(* CODESYS project METS_Software_Library.library
   Company: Marden Edwards LTD
   DefaultNamespace: LibB
   LanguageModelAttribute: qualified-access-only
   Title: METS_Software_Library
   Placeholder: LibA
   Version: 0.0.1

Project tree, tasks and I/O mapping:
  libraries: Tc2_Standard, * (Beckhoff Automation GmbH); Tc2_System, * (Beckhoff Automation GmbH); Tc2_Utilities, * (Beckhoff Automation GmbH)
  Maths/
    function F_Add [ST]
  Strings/
    Alias/
      data type T_Char
      data type T_LONGString
    Concat/
      function F_STRING_Concat3 [ST]
      function F_STRING_Concat4 [ST]
      function F_STRING_Concat5 [ST]
      function F_STRING_Concat6 [ST]
      function F_STRING_Concat7 [ST]
      function F_STRING_Concat8 [ST]
      function F_STRING_Concat9 [ST]
      function F_STRING_LongCONCAT [ST]
    Enumerations/
      data type E_STRING_ValidationCode
    Extract/
      function block FB_STRING_Extract [ST]
      function block FB_STRING_Extract_V2 [ST]
      function block FB_STRING_ExtractLong [ST]
    Manipulation/
      function F_STRING_AddPadding [ST]
      function F_STRING_AddPrefix [ST]
      function F_STRING_AddSuffix [ST]
      function F_STRING_CodeToHex [ST]
      function F_STRING_LongDELETE [ST]
      function F_STRING_LongFIND [ST]
      function F_STRING_LongLEFT [ST]
      function F_STRING_LongMID [ST]
      function F_STRING_LongRIGHT [ST]
      function F_STRING_ReplaceSingleChar [ST]
      function F_STRING_Wildcard [ST]
      function F_STRING_WriteEscapeCharacters [ST]
    Validation/
      function F_STRING_InvalidateASCIIChar [ST]
      function F_STRING_InvalidateNumericChar [ST]
      function F_STRING_IsNumber [ST]
      function F_STRING_Validate [ST]
      function F_STRING_ValidateCode [ST]
*)

// Strings/Alias/T_Char
TYPE T_Char : STRING(1); END_TYPE

// Strings/Alias/T_LONGString
TYPE T_LONGString : STRING(1024); END_TYPE

// Strings/Enumerations/E_STRING_ValidationCode
{attribute 'qualified_only'}
{attribute 'strict'}
{attribute 'to_string'}
TYPE E_STRING_ValidationCode :
(
	VALID := 0,
	EMPTY_STRING := 1,
	TOO_SHORT := 2,
	TOO_LONG := 3,
	INVALID := 4,
	INVALID_DECIMALPOINT := 5,
	MAXIMUM_LENGTH_EXCEEDED := 6
);
END_TYPE

// Maths/F_Add
FUNCTION F_Add : INT
VAR_INPUT
    nValue1 : INT;
    nValue2 : INT;
END_VAR

F_Add := nValue1 + nValue2;

END_FUNCTION

// Strings/Concat/F_STRING_Concat3
(* concatenate 3 strings *)
FUNCTION F_STRING_Concat3 : T_MaxString
VAR_INPUT
	sString1			: T_MaxString;		(* first string *)
	sString2			: T_MaxString;		(* second string *)
	sString3			: T_MaxString;		(* third string *)
END_VAR
VAR
END_VAR

F_STRING_Concat3 := CONCAT(sString1, sString2);
F_STRING_Concat3 := CONCAT(F_STRING_Concat3, sString3);

END_FUNCTION

// Strings/Concat/F_STRING_Concat4
(* concatenate 4 strings *)
FUNCTION F_STRING_Concat4 : T_MaxString
VAR_INPUT
	sString1			: T_MaxString;		(* first string *)
	sString2			: T_MaxString;		(* second string *)
	sString3			: T_MaxString;		(* third string *)
	sString4			: T_MaxString;		(* fourth string *)
END_VAR
VAR
END_VAR

F_STRING_Concat4 := CONCAT(sString1, sString2);
F_STRING_Concat4 := CONCAT(F_STRING_Concat4, sString3);
F_STRING_Concat4 := CONCAT(F_STRING_Concat4, sString4);

END_FUNCTION

// Strings/Concat/F_STRING_Concat5
(* concatenate 5 strings *)
FUNCTION F_STRING_Concat5 : T_MaxString
VAR_INPUT
	sString1			: T_MaxString;		(* first string *)
	sString2			: T_MaxString;		(* second string *)
	sString3			: T_MaxString;		(* third string *)
	sString4			: T_MaxString;		(* fourth string *)
	sString5			: T_MaxString;		(* fifth string *)
END_VAR
VAR
END_VAR

F_STRING_Concat5 := CONCAT(sString1, sString2);
F_STRING_Concat5 := CONCAT(F_STRING_Concat5, sString3);
F_STRING_Concat5 := CONCAT(F_STRING_Concat5, sString4);
F_STRING_Concat5 := CONCAT(F_STRING_Concat5, sString5);

END_FUNCTION

// Strings/Concat/F_STRING_Concat6
(* concatenate 6 strings *)
FUNCTION F_STRING_Concat6 : T_MaxString
VAR_INPUT
	sString1			: T_MaxString;		(* first string *)
	sString2			: T_MaxString;		(* second string *)
	sString3			: T_MaxString;		(* third string *)
	sString4			: T_MaxString;		(* fourth string *)
	sString5			: T_MaxString;		(* fifth string *)
	sString6			: T_MaxString;		(* sixth string *)
END_VAR
VAR
END_VAR

F_STRING_Concat6 := CONCAT(sString1, sString2);
F_STRING_Concat6 := CONCAT(F_STRING_Concat6, sString3);
F_STRING_Concat6 := CONCAT(F_STRING_Concat6, sString4);
F_STRING_Concat6 := CONCAT(F_STRING_Concat6, sString5);
F_STRING_Concat6 := CONCAT(F_STRING_Concat6, sString6);

END_FUNCTION

// Strings/Concat/F_STRING_Concat7
(* concatenate 7 strings *)
FUNCTION F_STRING_Concat7 : T_MaxString
VAR_INPUT
	sString1			: T_MaxString;		(* first string *)
	sString2			: T_MaxString;		(* second string *)
	sString3			: T_MaxString;		(* third string *)
	sString4			: T_MaxString;		(* fourth string *)
	sString5			: T_MaxString;		(* fifth string *)
	sString6			: T_MaxString;		(* sixth string *)
	sString7			: T_MaxString;		(* seventh string *)
END_VAR
VAR
END_VAR

F_STRING_Concat7 := CONCAT(sString1, sString2);
F_STRING_Concat7 := CONCAT(F_STRING_Concat7, sString3);
F_STRING_Concat7 := CONCAT(F_STRING_Concat7, sString4);
F_STRING_Concat7 := CONCAT(F_STRING_Concat7, sString5);
F_STRING_Concat7 := CONCAT(F_STRING_Concat7, sString6);
F_STRING_Concat7 := CONCAT(F_STRING_Concat7, sString7);

END_FUNCTION

// Strings/Concat/F_STRING_Concat8
(* concatenate 8 strings *)
FUNCTION F_STRING_Concat8 : T_MaxString
VAR_INPUT
	sString1			: T_MaxString;		(* first string *)
	sString2			: T_MaxString;		(* second string *)
	sString3			: T_MaxString;		(* third string *)
	sString4			: T_MaxString;		(* fourth string *)
	sString5			: T_MaxString;		(* fifth string *)
	sString6			: T_MaxString;		(* sixth string *)
	sString7			: T_MaxString;		(* seventh string *)
	sString8			: T_MaxString;		(* eigth string *)
END_VAR
VAR
END_VAR

F_STRING_Concat8 := CONCAT(sString1, sString2);
F_STRING_Concat8 := CONCAT(F_STRING_Concat8, sString3);
F_STRING_Concat8 := CONCAT(F_STRING_Concat8, sString4);
F_STRING_Concat8 := CONCAT(F_STRING_Concat8, sString5);
F_STRING_Concat8 := CONCAT(F_STRING_Concat8, sString6);
F_STRING_Concat8 := CONCAT(F_STRING_Concat8, sString7);
F_STRING_Concat8 := CONCAT(F_STRING_Concat8, sString8);

END_FUNCTION

// Strings/Concat/F_STRING_Concat9
(* concatenate 9 strings *)
FUNCTION F_STRING_Concat9 : T_MaxString
VAR_INPUT
	sString1			: T_MaxString;		(* first string *)
	sString2			: T_MaxString;		(* second string *)
	sString3			: T_MaxString;		(* third string *)
	sString4			: T_MaxString;		(* fourth string *)
	sString5			: T_MaxString;		(* fifth string *)
	sString6			: T_MaxString;		(* sixth string *)
	sString7			: T_MaxString;		(* seventh string *)
	sString8			: T_MaxString;		(* eigth string *)
	sString9			: T_MaxString;		(* ninth string *)
END_VAR
VAR
END_VAR
(*
-------------------------------------------------------------------------------------------------
Date		Version	Author	Comments
-------------------------------------------------------------------------------------------------
30/01/2015	3.00.00	PB		No change

-------------------------------------------------------------------------------------------------
05/02/2010	1.00.00	PB		Initial release

-------------------------------------------------------------------------------------------------
*)

F_STRING_Concat9 := CONCAT(sString1, sString2);
F_STRING_Concat9 := CONCAT(F_STRING_Concat9, sString3);
F_STRING_Concat9 := CONCAT(F_STRING_Concat9, sString4);
F_STRING_Concat9 := CONCAT(F_STRING_Concat9, sString5);
F_STRING_Concat9 := CONCAT(F_STRING_Concat9, sString6);
F_STRING_Concat9 := CONCAT(F_STRING_Concat9, sString7);
F_STRING_Concat9 := CONCAT(F_STRING_Concat9, sString8);
F_STRING_Concat9 := CONCAT(F_STRING_Concat9, sString9);

END_FUNCTION

// Strings/Concat/F_STRING_LongCONCAT
(* concatenate function for long strings *)
FUNCTION F_STRING_LongCONCAT : T_LongSTRING
VAR_INPUT
	sString1			: T_LongSTRING;		(* first string *)
	sString2			: T_LongSTRING;		(* second string *)
END_VAR
VAR
	_pPointer			: POINTER TO T_LongSTRING;		
	_nString1Length		: UINT;
	_nString2Length		: UINT;
END_VAR

(* length of 1st input string *)
_pPointer := ADR(sString1);
_nString1Length := TO_UINT(LEN2(_pPointer));

_pPointer := ADR(sString2);
(* max length of 2nd input string that can be handled without exceeding length of output string *)
_nString2Length := MIN(TO_UINT(LEN2(_pPointer)), SIZEOF(F_STRING_LongCONCAT) - _nString1Length - 1);

(* output string length <= 255 chars *)
IF _nString1Length + _nString2Length <= 255 THEN

	F_STRING_LongCONCAT := CONCAT(sString1, sString2);

(* output string length > 255 chars *)
ELSE

	(* string length > 0, must not call MEMMOVE with 0 bytes *)
	IF _nString1Length > 0 THEN

		(* move strString1 to output string *)
		MEMMOVE(ADR(F_STRING_LongCONCAT), ADR(sString1), _nString1Length);
		
	END_IF

	(* string length > 0, must not call MEMMOVE with 0 bytes *)
	IF _nString2Length > 0 THEN

		(* move strString2 to output string, clamp output if final length of string exceeds T_LongSTRING *)
		MEMMOVE(ADR(F_STRING_LongCONCAT) + _nString1Length, ADR(sString2), _nString2Length);
		
	END_IF

	(* reset last char to 16#00 to terminate the string with NULL *)
	MEMSET(ADR(F_STRING_LongCONCAT) + _nString1Length + _nString2Length, 16#00, 1);
	
END_IF

END_FUNCTION

// Strings/Extract/FB_STRING_Extract
(* extracts a substring defined by prefix and suffix *)
FUNCTION_BLOCK FB_STRING_Extract
VAR_INPUT
	bExtractData			: BOOL;			(* set TRUE to remove prefix and suffix from strData *)
	nExtractCharacters		: UINT;			(* if suffix is blank, number of data chars to extract *)
	sPrefix					: T_MaxString;	(* prefix string *)
	sSuffix					: T_MaxString;	(* suffix string *)
END_VAR
VAR_IN_OUT
	sString					: T_MaxString;	(* string to be searched *)
END_VAR
VAR_OUTPUT
	bStringFound			: BOOL;			(* TRUE = sub-string with matching prefix/suffix found *)
	nStartPosition			: UINT;			(* start pos of extracted string in sString *)
	sExtractedCharacters	: T_MaxString;	(* extracted data *)
END_VAR
VAR
	_nStringLength			: UINT;
	_nPrefixLength			: UINT;
	_nSuffixLength			: UINT;
	_nEndPosition			: UINT;
	_bStartPositionFound	: BOOL;
	_bEndPositionFound		: BOOL;
	_nCharacters			: UINT;
	_nMaxIndex				: UINT;
	_nIndex					: UINT;
END_VAR

(* calc string lengths *)
_nStringLength := INT_TO_UINT(LEN(sString));
_nPrefixLength := INT_TO_UINT(LEN(sPrefix));
_nSuffixLength := INT_TO_UINT(LEN(sSuffix));

(* string to be searched is not empty and prefix or suffix or no or chars to extract is defined *)
IF _nStringLength > 0 AND (_nPrefixLength > 0 OR _nSuffixLength > 0 OR nExtractCharacters > 0) THEN

	(* clear outputs *)
	bStringFound := FALSE;
	_nCharacters := 0;
	nStartPosition := 0;
	sExtractedCharacters := '';

	(* initialise char index values *)
	_bStartPositionFound := FALSE;
	_bEndPositionFound := FALSE;
	_nEndPosition := 0;

	(* max search index, based on string length - 1 due to starting at 0 and length of prefix *)
	_nMaxIndex := (_nStringLength - 1) + (_nPrefixLength - 1);

	(* for each character in the string *)
	FOR _nIndex := 0 TO _nMaxIndex DO

		(* prefix has not been found *)
		IF _bStartPositionFound = FALSE THEN

			(* no prefix defined  *)
			IF _nPrefixLength = 0 THEN

				(* start at beginning if string *)
				nStartPosition := 1;
				_bStartPositionFound := TRUE;

			(* prefix defined  *)
			ELSE

				(* compare partial string with prefix *)
				IF MEMCMP(ADR(sString) + _nIndex, ADR(sPrefix), _nPrefixLength) = 0 THEN

					(* prefix position found *)
					nStartPosition := _nIndex + 1;
					_bStartPositionFound := TRUE;

					(* skip to end of prefix to continue search *)
					_nIndex := _nIndex + _nPrefixLength - 1;
					
				END_IF
				
			END_IF

		(* suffix has not been found *)
		ELSIF _bEndPositionFound = FALSE THEN

			(* no suffix defined  *)
			IF _nSuffixLength = 0 THEN

				(* start at 1st char of string *)
				_bEndPositionFound := TRUE;

				(* calculate end position *)
				_nEndPosition := MIN((nStartPosition - 1) + nExtractCharacters + _nPrefixLength, _nStringLength);

			(* suffix defined  *)
			ELSE

				(* compare partial string with suffix *)
				IF MEMCMP(ADR(sString) + _nIndex, ADR(sSuffix), _nSuffixLength) = 0 THEN

					(* suffix position found, calculate end position *)
					_nEndPosition := _nIndex + _nSuffixLength;
					_bEndPositionFound := TRUE;

					(* no prefix defined and number of chars to extract is defined *)
					IF _nPrefixLength = 0 AND nExtractCharacters > 0 THEN

						(* re-calculate start position *)
						nStartPosition := MAX(_nEndPosition - nExtractCharacters - 1, 1);
						
					END_IF

					(* search complete, quit FOR loop *)
					EXIT;
					
				END_IF
				
			END_IF

		(* prefix and suffix found *)
		ELSE

			(* quit FOR loop *)
			EXIT;
			
		END_IF
		
	END_FOR

	(* start and end positions known *)
	IF _bStartPositionFound = TRUE AND _bEndPositionFound = TRUE THEN

		(* string has been found *)
		bStringFound := TRUE;

		(* return string without prefix and suffix *)
		IF bExtractData = TRUE THEN

			(* total chars to be moved to strData *)
			_nCharacters := (_nEndPosition - (nStartPosition - 1)) - _nPrefixLength - _nSuffixLength;

			(* 1 or more chars to be moved *)
			IF _nCharacters > 0 THEN

				(* move data to sResult *)
				MEMMOVE(ADR(sExtractedCharacters), ADR(sString) + (nStartPosition - 1) + _nPrefixLength, _nCharacters);
				
			END_IF

		(* return string with prefix and suffix *)
		ELSE

			(* total chars to be moved to strData *)
			_nCharacters := _nEndPosition - (nStartPosition - 1);

			(* 1 or more chars to be moved *)
			IF _nCharacters > 0 THEN

				(* move data to sResult *)
				MEMMOVE(ADR(sExtractedCharacters), ADR(sString) + (nStartPosition - 1), _nCharacters);
				
			END_IF
			
		END_IF

		(* terminate sResult *)
		MEMSET(ADR(sExtractedCharacters) + _nCharacters, 16#00, 1);

		(* 1 or more chars after strSuffix *)
		IF _nStringLength > (_nEndPosition - (nStartPosition - 1)) THEN

			(* shift post-suffix chars to prefix position *)
			MEMMOVE(ADR(sString) + (nStartPosition - 1), ADR(sString) + _nEndPosition, _nStringLength - (_nEndPosition - (nStartPosition - 1)));
			
		END_IF

		(* terminate strString *)
		MEMSET(ADR(sString) + _nStringLength - (_nEndPosition - (nStartPosition - 1)), 16#00, 1);
		
	END_IF

(* string to be searched is empty or prefix and suffix and both blank *)
ELSE

	(* clear outputs *)
	bStringFound := FALSE;
	_nCharacters := 0;
	sExtractedCharacters := '';
	
END_IF

END_FUNCTION_BLOCK

// Strings/Extract/FB_STRING_Extract_V2
(* extracts a substring defined by prefix and suffix *)
FUNCTION_BLOCK FB_STRING_Extract_V2
VAR_INPUT
	bIgnoreCase				: BOOL;
	sPrefix					: STRING(10);	(* prefix string *)
	sSuffix					: STRING(10);	(* suffix string *)
	nExtractCharacters		: BYTE;			(* if suffix is blank, >0 = no of chars to extract , 0 = remainder of string *)
END_VAR
VAR_IN_OUT
	sString					: T_MaxString;	(* string to be searched *)
END_VAR
VAR_OUTPUT
	bStringFound			: BOOL;			(* TRUE = sub-string with matching prefix/suffix found *)
	nCharactersFound		: UINT;			(* no of chars in sub-string *)
	sExtractedCharacters	: T_MaxString;	(* sub-string with prefix and suffix *)
END_VAR
VAR
	_nPrefixPosition		: UINT;
	_nSuffixPosition		: UINT;
	_nIndex					: UINT;
	_sStringInternal		: T_MaxString;
	_sPrefixInternal		: STRING(10);
	_sSuffixInternal		: STRING(10);
	_sCheckString			: STRING(10);
END_VAR

(* string to be searched is not empty *)
IF LEN(sString) > 0 THEN

	(* matching for Prefix and Suffix is case-sesnsitive *)
	IF bIgnoreCase = FALSE THEN

		(* internal comparators are not changed *)
		_sStringInternal := sString;
		_sPrefixInternal := sPrefix;
		_sSuffixInternal := sSuffix;

	(* ignore case when matching for Prefix and Suffix *)
	ELSE

		(* internal comparators are all converted to lower case *)
		_sStringInternal := F_ToLCase(sString);
		_sPrefixInternal := F_ToLCase(sPrefix);
		_sSuffixInternal := F_ToLCase(sSuffix);
		
	END_IF

	(* prefix is blank *)
	IF _sPrefixInternal = '' THEN

		(* start at beginning of string *)
		_nPrefixPosition := 1;

	(* prefix is not blank *)
	ELSE

		(* find 1st occurrence of prefix in strString *)
		_nPrefixPosition := FIND(_sStringInternal, _sPrefixInternal);
		
	END_IF

	(* suffix is blank *)
	IF _sSuffixInternal = '' THEN
	
		(* no of chars not specified *)
		IF nExtractCharacters = 0 THEN
	
			(* finish at end of string *)
			_nSuffixPosition := LEN(_sStringInternal);
	
		(* no of chars specified *)
		ELSE
	
			(* finish at end of string *)
			_nSuffixPosition := _nPrefixPosition + nExtractCharacters - 1;
			
		END_IF
	
	(* suffix is not blank *)
	ELSE
	
		_nSuffixPosition := 0;
	
		(* find 1st occurrence of suffix in strString AFTER position of strPrefix *)
		FOR _nIndex := _nPrefixPosition + LEN(_sPrefixInternal) TO LEN(_sStringInternal) DO
	
			(* extract string same length as suffix string *)
			_sCheckString := MID(_sStringInternal, LEN(_sSuffixInternal), _nIndex);
	
			(* extracted string = suffix string *)
			IF _sCheckString = _sSuffixInternal THEN
	
				(* position of suffix string *)
				_nSuffixPosition := _nIndex;
				EXIT;
				
			END_IF
			
		END_FOR
		
	END_IF
	
	
	(* prefix and suffix both exist *)
	IF _nPrefixPosition > 0 AND _nSuffixPosition > 0 THEN
	
		(* extract sub-string *)
		sExtractedCharacters := MID(sString, _nSuffixPosition + MAX(LEN(_sSuffixInternal), 1) - _nPrefixPosition, _nPrefixPosition);

		(* delete sub-string *)
		sString := DELETE(sString, _nSuffixPosition + MAX(LEN(_sSuffixInternal), 1) - _nPrefixPosition, _nPrefixPosition);
	
		(* update outputs *)
		bStringFound := TRUE;
		nCharactersFound := LEN(sExtractedCharacters);
	
	(* no prefix or suffix defined, cannot search for string *)
	ELSE
	
		sExtractedCharacters := '';
		bStringFound := FALSE;
		nCharactersFound := 0;
		
	END_IF

(* string to be searched is empty *)
ELSE

	(* reset outputs *)
	bStringFound := FALSE;
	nCharactersFound := 0;
	sExtractedCharacters := '';
	
END_IF

END_FUNCTION_BLOCK

// Strings/Extract/FB_STRING_ExtractLong
(* extracts a substring from a long string defined by prefix and suffix *)
FUNCTION_BLOCK FB_STRING_ExtractLong
VAR_INPUT
	bExtractData			: BOOL;			(* set TRUE to remove prefix and suffix from strData *)
	nExtractCharacters		: UINT;			(* if suffix is blank, number of data chars to extract *)
	sPrefix					: T_MaxString;	(* prefix string *)
	sSuffix					: T_MaxString;	(* suffix string *)
END_VAR
VAR_IN_OUT
	sString					: T_LongSTRING;	(* string to be searched *)
END_VAR
VAR_OUTPUT
	bStringFound			: BOOL;			(* TRUE = sub-string with matching prefix/suffix found *)
	nStartPosition			: UINT;			(* start pos of extracted string in strString *)
	sExtractedCharacters	: T_LongSTRING;	(* extracted data *)
END_VAR
VAR
	_bStartPositionFound	: BOOL;
	_bEndPositionFound		: BOOL;
	_nStringLength			: UINT;
	_nPrefixLength			: UINT;
	_nSuffixLength			: UINT;
	_nEndPosition			: UINT;
	_nCharacters			: UINT;
	_nMaxIndex				: UINT;
	_nIndex					: UINT;
END_VAR

(* calc string lengths *)
_nStringLength := UDINT_TO_UINT(LEN2(ADR(sString)));
_nPrefixLength := INT_TO_UINT(LEN(sPrefix));
_nSuffixLength := INT_TO_UINT(LEN(sSuffix));

(* string to be searched is not empty and prefix or suffix or no or chars to extract is defined *)
IF _nStringLength > 0 AND (_nPrefixLength > 0 OR _nSuffixLength > 0 OR nExtractCharacters > 0) THEN

	(* clear outputs *)
	bStringFound := FALSE;
	_nCharacters := 0;
	nStartPosition := 0;
	sExtractedCharacters := '';

	(* initialise char index values *)
	_bStartPositionFound := FALSE;
	_bEndPositionFound := FALSE;
	_nEndPosition := 0;

	(* max search index, based on string length - 1 due to starting at 0 and length of prefix *)
	_nMaxIndex := (_nStringLength - 1) + (_nPrefixLength - 1);

	(* for each character in the string *)
	FOR _nIndex := 0 TO _nMaxIndex DO

		(*IF nIndex = nMaxIndex  AND NOT bStartPosFound THEN

			strString :='1';

		(* prefix has not been found *)
		ELS*)IF _bStartPositionFound = FALSE THEN

			(* no prefix defined  *)
			IF _nPrefixLength = 0 THEN

				(* start at beginning if string *)
				nStartPosition := 1;
				_bStartPositionFound := TRUE;

			(* prefix defined  *)
			ELSE

				(* compare partial string with prefix *)
				IF MEMCMP(ADR(sString) + _nIndex, ADR(sPrefix), _nPrefixLength) = 0 THEN

					(* prefix position found *)
					nStartPosition := _nIndex + 1;
					_bStartPositionFound := TRUE;

					(* skip to end of prefix to continue search *)
					_nIndex := _nIndex + _nPrefixLength - 1;
					
				END_IF
				
			END_IF

		(* suffix has not been found *)
		ELSIF _bEndPositionFound = FALSE THEN

			(* no suffix defined  *)
			IF _nSuffixLength = 0 THEN

				(* start at 1st char of string *)
				_bEndPositionFound := TRUE;

				(* calculate end position *)
				_nEndPosition := MIN((nStartPosition - 1) + nExtractCharacters + _nPrefixLength, _nStringLength);

			(* suffix defined  *)
			ELSE

				(* compare partial string with suffix *)
				IF MEMCMP(ADR(sString) + _nIndex, ADR(sSuffix), _nSuffixLength) = 0 THEN

					(* suffix position found, calculate end position *)
					_nEndPosition := _nIndex + _nSuffixLength;
					_bEndPositionFound := TRUE;

					(* no prefix defined and number of chars to extract is defined *)
					IF _nPrefixLength = 0 AND nExtractCharacters > 0 THEN

						(* re-calculate start position *)
						nStartPosition := MAX(_nEndPosition - nExtractCharacters - 1, 1);
						
					END_IF

					(* search complete, quit FOR loop *)
					EXIT;
					
				END_IF
				
			END_IF

		(* prefix and suffix found *)
		ELSE

			(* quit FOR loop *)
			EXIT;

		END_IF
		
	END_FOR

	(* start and end positions known *)
	IF _bStartPositionFound = TRUE AND _bEndPositionFound = TRUE THEN

		(* string has been found *)
		bStringFound := TRUE;

		(* return string without prefix and suffix *)
		IF bExtractData = TRUE THEN

			(* total chars to be moved to strData *)
			_nCharacters := (_nEndPosition - (nStartPosition - 1)) - _nPrefixLength - _nSuffixLength;

			(* 1 or more chars to be moved *)
			IF _nCharacters > 0 THEN

				(* move data to strData *)
				MEMMOVE(ADR(sExtractedCharacters), ADR(sString) + (nStartPosition - 1) + _nPrefixLength, _nCharacters);
				
			END_IF

		(* return string with prefix and suffix *)
		ELSE

			(* total chars to be moved to strData *)
			_nCharacters := _nEndPosition - (nStartPosition - 1);

			(* 1 or more chars to be moved *)
			IF _nCharacters > 0 THEN

				(* move data to strData *)
				MEMMOVE(ADR(sExtractedCharacters), ADR(sString) + (nStartPosition - 1), _nCharacters);
				
			END_IF
			
		END_IF

		(* terminate strData *)
		MEMSET(ADR(sExtractedCharacters) + _nCharacters, 16#00, 1);

		(* 1 or more chars after strSuffix *)
		IF _nStringLength> (_nEndPosition - (nStartPosition - 1)) THEN

			(* shift post-suffix chars to prefix position *)
			MEMMOVE(ADR(sString) + (nStartPosition - 1), ADR(sString) + _nEndPosition, _nStringLength - (_nEndPosition - (nStartPosition - 1)));
			
		END_IF

		(* terminate strString *)
		MEMSET(ADR(sString) + _nStringLength - (_nEndPosition - (nStartPosition - 1)), 16#00, 1);
		
	END_IF

(* string to be searched is empty or prefix and suffix and both blank *)
ELSE

	(* clear outputs *)
	bStringFound := FALSE;
	_nCharacters := 0;
	sExtractedCharacters := '';
	
END_IF

END_FUNCTION_BLOCK

// Strings/Manipulation/F_STRING_AddPadding
(* Adds leading '0' to a given string returning it as a string.  Number has to be a positive integer *)
FUNCTION F_STRING_AddPadding : STRING 		(* String with leading '0' applied.  Max length 80 characters *)
VAR_INPUT
	nNumber				: UDINT;			(* Number to add leading '0' to *)
	nSize				: UINT;				(* Total size of the returning string including the original number *)
END_VAR
VAR
	_Size				: UINT;
	_sTemp				: STRING;
END_VAR

IF nSize > 80 THEN 

	_sTemp := UDINT_TO_STRING(nNumber);
	F_STRING_AddPadding := _sTemp;

ELSE

	_Size := nSize;
	_sTemp := UDINT_TO_STRING(nNumber);
	
	WHILE LEN(_sTemp) < _Size DO

		_sTemp := CONCAT('0',_sTemp);

	END_WHILE
	
	F_STRING_AddPadding := _sTemp;

END_IF

END_FUNCTION

// Strings/Manipulation/F_STRING_AddPrefix
(* add specified char(s) in front of a string to make up to specified length *)
FUNCTION F_STRING_AddPrefix : T_MaxString
VAR_INPUT
	sString				: T_MaxString;	(* initial string *)
	nTargetLength 		: UINT;			(* total string length required *)
	sCharacterToAppend	: T_Char;		(* character to be inserted at start of the string *)
END_VAR
VAR
	_nStringLength		: UINT;
	_nCharactersRequired: UINT; 
END_VAR

(* length of input string *)
_nStringLength := TO_UINT(LEN(sString));

(* total prefix chars required *)
_nCharactersRequired := MIN(nTargetLength, SIZEOF(F_STRING_AddPrefix) - 1) - _nStringLength;

(* string needs additional chars *)
IF _nCharactersRequired > 0 THEN

	(* set prefix chars to specified character *)
	MEMSET(ADR(F_STRING_AddPrefix), F_ToASC(sCharacterToAppend), _nCharactersRequired);

	(* append strString to output string *)
	MEMMOVE(ADR(F_STRING_AddPrefix) + _nCharactersRequired, ADR(sString), _nStringLength);

	(* reset last char to 16#00 to terminate the string *)
	MEMSET(ADR(F_STRING_AddPrefix) + _nCharactersRequired + _nStringLength, 16#00, 1);

(* no additional chars required *)
ELSE

	(* copy strString to output *)
	F_STRING_AddPrefix := sString;
	
END_IF

END_FUNCTION

// Strings/Manipulation/F_STRING_AddSuffix
(* add specified char(s) to the end of a string to make up to specified length *)
FUNCTION F_STRING_AddSuffix : T_MaxString
VAR_INPUT
	sString				: T_MaxString;	(* initial string *)
	nTargetLength 		: UINT;			(* string length required *)
	sCharacterToAppend	: T_Char;		(* character to be appended to the string *)
END_VAR
VAR
	_nStringLength		: UINT;
	_nCharactersRequired: UINT;
END_VAR

(* length of input string *)
_nStringLength := TO_UINT(LEN(sString));

(* total suffix chars required *)
_nCharactersRequired := MIN(nTargetLength, SIZEOF(F_STRING_AddSuffix) - 1) - _nStringLength;

(* string needs additional chars *)
IF _nCharactersRequired > 0 THEN

	(* append strString to output string *)
	MEMMOVE(ADR(F_STRING_AddSuffix), ADR(sString), _nStringLength);

	(* set prefix chars to specified character *)
	MEMSET(ADR(F_STRING_AddSuffix) + _nStringLength, F_ToASC(sCharacterToAppend), _nCharactersRequired);

	(* reset last char to 16#00 to terminate the string *)
	MEMSET(ADR(F_STRING_AddSuffix) + _nStringLength + _nCharactersRequired, 16#00, 1);

(* no additional chars required *)
ELSE

	(* copy strString to output *)
	F_STRING_AddSuffix := sString;
END_IF

END_FUNCTION

// Strings/Manipulation/F_STRING_CodeToHex
(* Takes a string and returns as a string of hexcodes *)
FUNCTION F_STRING_CodeToHex : T_MaxString
VAR_INPUT
	sCode				: T_MaxString;
END_VAR
VAR
	_nCharacterIndex	: UINT;
	_sCharacter			: STRING(1);
	_nCharacterInDec	: BYTE;
	_sCharacterInHex	: STRING(2);
END_VAR

(* reset output *)
F_STRING_CodeToHex := '';

(* Make sure there is a string to process *)
IF LEN(sCode)  > 0  AND LEN(sCode) < 256 THEN

	(* check each character in the code *)
	FOR _nCharacterIndex := 1 TO LEN(sCode)  DO

		(* get next character from the string *)
		_sCharacter := MID(sCode, 1, _nCharacterIndex);
		_nCharacterInDec := F_ToASC(_sCharacter);
		_sCharacterInHex := DATA_TO_HEXSTR(ADR(_nCharacterInDec), SIZEOF(_nCharacterInDec), FALSE);
		F_STRING_CodeToHex := CONCAT(F_STRING_CodeToHex, _sCharacterInHex);
		
	END_FOR

ELSIF LEN(sCode) >= 256 THEN
	
	F_STRING_CodeToHex :='Exceed_String_Length';
	
END_IF

END_FUNCTION

// Strings/Manipulation/F_STRING_LongDELETE
(* DELETE function for long string *)
FUNCTION F_STRING_LongDELETE : T_LongSTRING
VAR_INPUT
	sString				: T_LongSTRING;
	nNumOfCharsToDelete	: UINT;	(* number of characters to delete *)
	nPosition			: UINT;	(* 1st character to delete *)
END_VAR
VAR
	_pPointer			: POINTER TO T_LongSTRING;
	_nStringLength		: UINT;
END_VAR

(* length of input string *)
_pPointer := ADR(sString);
_nStringLength := TO_UINT(LEN2(_pPointer));

(* input string length <= 255 chars *)
IF _nStringLength <= 255 THEN

	(* use standard DELETE function *)
	F_STRING_LongDELETE := DELETE(sString, TO_INT(nNumOfCharsToDelete), TO_INT(nPosition));

(* input string length > 255 chars *)
ELSE

	(* no of chars specified, 1st char is specified and 1st char is present in string *)
	IF nNumOfCharsToDelete > 0 AND nPosition > 0 AND nPosition <= _nStringLength THEN

		(* string contains chars before DELETE range *)
		IF nPosition > 1 THEN

			(* copy chars before DELETE range to output *)
			MEMMOVE(ADR(F_STRING_LongDELETE), ADR(sString), nPosition - 1);
		END_IF

		(* string contains chars after DELETE range *)
		IF _nStringLength > nPosition + nNumOfCharsToDelete - 1 THEN

			(* copy chars after DELETE range to output *)
			MEMMOVE(ADR(F_STRING_LongDELETE) + nPosition - 1, ADR(sString) + nPosition + nNumOfCharsToDelete - 1,  _nStringLength - (nPosition + nNumOfCharsToDelete - 1));
		END_IF

		(* set last char to 16#00 to terminate the string with NULL *)
		MEMSET(ADR(F_STRING_LongDELETE) + _nStringLength - nNumOfCharsToDelete, 16#00, 1);

	(* no of chars not specified, 1st char not speciifed or 1st char does not exist in string *)
	ELSE

		(* pass input string unmodified *)
		F_STRING_LongDELETE := sString;
		
	END_IF
	
END_IF

END_FUNCTION

// Strings/Manipulation/F_STRING_LongFIND
(* FIND function for long string *)
FUNCTION F_STRING_LongFIND : UINT
VAR_INPUT
	sString					: T_LongSTRING;
	sSearchString			: T_LongSTRING;	(* search string *)
END_VAR
VAR
	_pPointer				: POINTER TO T_LongSTRING;
	_nStringLength			: UINT;
	_nSearchStringLength	: UINT;
	_nIndex					: UINT;
END_VAR

(* get lengths of both strings *)
_pPointer := ADR(sString);
_nStringLength := TO_UINT(LEN2(_pPointer));
_pPointer := ADR(sSearchString);
_nSearchStringLength := TO_UINT(LEN2(_pPointer));

(* strString1 and strString2 are 255 chars or less *)
IF _nStringLength <= 255 AND _nSearchStringLength <= 255 THEN

	(* use standard FIND function *)
	F_STRING_LongFIND := TO_UINT(FIND(sString, sSearchString));

(* strString1 string length > 255 chars *)
ELSE

	(* String1 is at least as long as String2 and String2 contains data *)
	IF _nStringLength >= _nSearchStringLength AND _nSearchStringLength > 0 THEN

		(* for each char in source string *)
		FOR _nIndex := 0 TO _nStringLength - _nSearchStringLength DO

			(* compare source data with search string *)
			IF MEMCMP(ADR(sString) + _nIndex, ADR(sSearchString), _nSearchStringLength) = 0 THEN

				(* match found, return index where 1st char of matching string was found *)
				F_STRING_LongFIND := _nIndex + 1;
				
				EXIT;
				
			END_IF
			
		END_FOR

	(* invalid input strings *)
	ELSE

		(* string not found *)
		F_STRING_LongFIND := 0;
		
	END_IF
	
END_IF

END_FUNCTION

// Strings/Manipulation/F_STRING_LongLEFT
(* LEFT function for long string *)
FUNCTION F_STRING_LongLEFT : T_LongSTRING
VAR_INPUT
	sString				: T_LongSTRING;
	nLength				: UINT;	(* number of characters to extract *)
END_VAR
VAR
	_pPointer			: POINTER TO T_LongSTRING;	
	_nStringLength		: UINT;
	_nActualLength		: UINT;
END_VAR

(* length of input string *)
_pPointer := ADR(sString);
_nStringLength := TO_UINT(LEN2(_pPointer));

(* input string length <= 255 chars *)
IF _nStringLength <= 255 THEN

	(* use standard LEFT function *)
	F_STRING_LongLEFT := LEFT(sString, nLength);

(* input string length > 255 chars *)
ELSE

	(* no of chars specified *)
	IF nLength > 0 AND _nStringLength > 0 THEN

		(* chars required < strString length *)
		IF nLength < _nStringLength THEN

			(* clamp no of chars to be extracted to length of input string *)
			_nActualLength := MIN(nLength, _nStringLength);
	
			(* extract chars from strString *)
			MEMMOVE(ADR(F_STRING_LongLEFT), ADR(sString), _nActualLength);
	
			(* set last char to 16#00 to terminate the string with NULL *)
			MEMSET(ADR(F_STRING_LongLEFT) + _nActualLength, 16#00, 1);

		(* chars required >= strString length *)
		ELSE

			(* return complete string *)
			F_STRING_LongLEFT := sString;
			
		END_IF

	(* no length specified *)
	ELSE

		(* return empty string *)
		F_STRING_LongLEFT := '';
		
	END_IF
	
END_IF

END_FUNCTION

// Strings/Manipulation/F_STRING_LongMID
(* MID function for long string *)
FUNCTION F_STRING_LongMID : T_LongSTRING
VAR_INPUT
	sString				: T_LongSTRING;
	nNumCharsToExtract	: UINT;	(* number of characters to extract *)
	nPosition			: UINT;	(* 1st character to extract *)
END_VAR
VAR
	_pPointer			: POINTER TO T_LongSTRING;	
	_nStringLength		: UINT;
END_VAR

(* length of input string *)
_pPointer := ADR(sString);
_nStringLength := TO_UINT(LEN2(_pPointer));

(* input string length <= 255 chars *)
IF _nStringLength <= 255 THEN

	(* use standard MID function *)
	F_STRING_LongMID := MID(sString, nNumCharsToExtract, nPosition);

(* input string length > 255 chars *)
ELSE

	(* no of chars specified, 1st char is specified and 1st char is present in string *)
	IF nNumCharsToExtract > 0 AND nPosition > 0 AND nPosition <= _nStringLength THEN

		(* extract chars from strString *)
		MEMMOVE(ADR(F_STRING_LongMID), ADR(sString) + nPosition - 1, nNumCharsToExtract);

		(* set last char to 16#00 to terminate the string with NULL *)
		MEMSET(ADR(F_STRING_LongMID) + nNumCharsToExtract, 16#00, 1);

	(* no of chars not specified, 1st char not speciifed or 1st char does not exist in string *)
	ELSE

		(* clear output *)
		F_STRING_LongMID := '';
		
	END_IF
	
END_IF

END_FUNCTION

// Strings/Manipulation/F_STRING_LongRIGHT
(* RIGHT function for long string *)
FUNCTION F_STRING_LongRIGHT : T_LongSTRING
VAR_INPUT
	sString				: T_LongSTRING;
	nNumCharsToExtract	: UINT;	(* number of characters to extract *)
END_VAR
VAR
	_pPointer			: POINTER TO T_LongSTRING;	
	_nStringLength		: UINT;
	_nActualLength		: UINT;
END_VAR

(* length of input string *)
_pPointer := ADR(sString);
_nStringLength := TO_UINT(LEN2(_pPointer));

(* input string length <= 255 chars *)
IF _nStringLength <= 255 THEN

	(* use standard RIGHT function *)
	F_STRING_LongRIGHT := RIGHT(sString, nNumCharsToExtract);

(* input string length > 255 chars *)
ELSE

	(* no of chars specified *)
	IF nNumCharsToExtract > 0 AND _nStringLength > 0 THEN

		(* chars required < strString length *)
		IF nNumCharsToExtract < _nStringLength THEN

			(* clamp no of chars to be extracted to length of input string *)
			_nActualLength := MIN(nNumCharsToExtract, _nStringLength);

			(* extract chars from strString *)
			MEMMOVE(ADR(F_STRING_LongRIGHT), ADR(sString) + _nStringLength - _nActualLength, _nActualLength);

			(* set last char to 16#00 to terminate the string with NULL *)
			MEMSET(ADR(F_STRING_LongRIGHT) + _nActualLength, 16#00, 1);

		(* chars required >= strString length *)
		ELSE

			(* return complete string *)
			F_STRING_LongRIGHT := sString;
			
		END_IF

	(* no chars specified *)
	ELSE

		(* return empty string *)
		F_STRING_LongRIGHT := '';
		
	END_IF
	
END_IF

END_FUNCTION

// Strings/Manipulation/F_STRING_ReplaceSingleChar
(* searches for and replaces a character with a new one *)
FUNCTION F_STRING_ReplaceSingleChar : T_MaxString
VAR_INPUT
	sString				: T_MAXString;		(* Search string *)
	sCharacterToRemove	: T_Char := '$1D';	(* Character to search for and remove *)
	sReplacmentCharacter: T_Char := '';		(* Character to replace *)
END_VAR
VAR
END_VAR

(* reset output *)
F_STRING_ReplaceSingleChar :='';

WHILE FIND(sString, sCharacterToRemove) > 0 DO
	sString := REPLACE(sString,sReplacmentCharacter, LEN(sCharacterToRemove), FIND(sString, sCharacterToRemove));
END_WHILE

F_STRING_ReplaceSingleChar	:= sString;

END_FUNCTION

// Strings/Manipulation/F_STRING_Wildcard
(* replaces date and time wildcards in string *)
FUNCTION F_STRING_Wildcard : T_MaxString
VAR_INPUT
	sString				: T_MaxString;	(* string with wildcard markers *)
	stDateTime			: TIMESTRUCT;	(* date/time structure *)
END_VAR
VAR
	_fbExtractData		: FB_STRING_Extract;
	_sWildcard			: T_MaxString;
	_sData				: STRING(4);
	_nCharacterPosition	: UINT;
END_VAR
VAR CONSTANT
	arrMonthCode	: ARRAY[0..12] OF STRING(1) :=[ '', 'A', 'B', 'C', 'D', 'E', 'F', 'G', 'H', 'I', 'J', 'K', 'L'];
END_VAR
(*
The following wildcard strings are supported:
YYYY - Year (4 chars)				hh	- hour
YY	 - Year (last 2 chars)			mm	- minute
Y	 - Year (last char only)		ss	- second
MM	 - Month (01-12 = Jan-Dec)		t	- tenth of second
M	 - Month (A-L = Jan-Dec)
DD	 - Date
*)

(* find and extract wildcard string, enclosed by '#' chars *)
_fbExtractData(
	bExtractData		:= TRUE,
	nExtractCharacters	:= 0,
	sPrefix			:= '#',
	sSuffix			:= '#',
	sString			:= sString
);

(* wildcard string found *)
IF _fbExtractData.bStringFound = TRUE THEN

	(* log wildcard string for modification *)
	_sWildcard := _fbExtractData.sExtractedCharacters;

	(* check for wildcard 'YYYY' *)
	_nCharacterPosition := FIND(_sWildcard, 'YYYY');
	IF _nCharacterPosition > 0 THEN

		(* generate year as 4 chars and replace YYYY *)
		_sData := F_STRING_AddPrefix(WORD_TO_STRING(stDateTime.wYear), 4, '0');
		_sWildcard := REPLACE(_sWildcard, _sData, 4, _nCharacterPosition);

	(* wildcard 'YYYY' not found *)
	ELSE

		(* check for wildcard 'YY' *)
		_nCharacterPosition := FIND(_sWildcard, 'YY');
		IF _nCharacterPosition > 0 THEN

			(* generate year as 2 chars and replace YY *)
			_sData := F_STRING_AddPrefix(RIGHT(WORD_TO_STRING(stDateTime.wYear), 2), 2, '0');
			_sWildcard := REPLACE(_sWildcard, _sData, 2, _nCharacterPosition);

		(* wildcard 'YY' not found *)
		ELSE
	
			(* check for wildcard 'Y' *)
			_nCharacterPosition := FIND(_sWildcard, 'Y');
			IF _nCharacterPosition > 0 THEN
	
				(* generate year as 1 char and replace Y *)
				_sData := RIGHT(WORD_TO_STRING(stDateTime.wYear), 1);
				_sWildcard := REPLACE(_sWildcard, _sData, 1, _nCharacterPosition);
			END_IF
		END_IF
	END_IF

	(* check for wildcard 'DD' *)
	_nCharacterPosition := FIND(_sWildcard, 'DD');
	IF _nCharacterPosition > 0 THEN

		(* generate date as 2 chars and replace DD *)
		_sData := F_STRING_AddPrefix(WORD_TO_STRING(stDateTime.wDay), 2, '0');
		_sWildcard := REPLACE(_sWildcard, _sData, 2, _nCharacterPosition);
	END_IF

	(* check for wildcard 'hh' *)
	_nCharacterPosition := FIND(_sWildcard, 'hh');
	IF _nCharacterPosition > 0 THEN

		(* generate hour as 2 chars and replace hh *)
		_sData := F_STRING_AddPrefix(WORD_TO_STRING(stDateTime.wHour), 2, '0');
		_sWildcard := REPLACE(_sWildcard, _sData, 2, _nCharacterPosition);
	END_IF

	(* check for wildcard 'mm' *)
	_nCharacterPosition := FIND(_sWildcard, 'mm');
	IF _nCharacterPosition > 0 THEN

		(* generate minute as 2 chars and replace mm *)
		_sData := F_STRING_AddPrefix(WORD_TO_STRING(stDateTime.wMinute), 2, '0');
		_sWildcard := REPLACE(_sWildcard, _sData, 2, _nCharacterPosition);
	END_IF

	(* check for wildcard 'ss' *)
	_nCharacterPosition := FIND(_sWildcard, 'ss');
	IF _nCharacterPosition > 0 THEN

		(* generate second as 2 chars and replace ss *)
		_sData := F_STRING_AddPrefix(WORD_TO_STRING(stDateTime.wSecond), 2, '0');
		_sWildcard := REPLACE(_sWildcard, _sData, 2, _nCharacterPosition);
	END_IF

	(* check for wildcard 't' *)
	_nCharacterPosition := FIND(_sWildcard, 't');
	IF _nCharacterPosition > 0 THEN

		(* generate tenth of second as 1 char and replace t *)
		_sData := WORD_TO_STRING(stDateTime.wMilliseconds / 100);
		_sWildcard := REPLACE(_sWildcard, _sData, 1, _nCharacterPosition);
	END_IF

	(* check for wildcard 'MM' *)
	_nCharacterPosition := FIND(_sWildcard, 'MM');
	IF _nCharacterPosition > 0 THEN

		(* generate month as 2 chars and replace MM *)
		_sData := F_STRING_AddPrefix(WORD_TO_STRING(stDateTime.wMonth), 2, '0');
		_sWildcard := REPLACE(_sWildcard, _sData, 2, _nCharacterPosition);

	(* wildcard 'YYYY' not found *)
	ELSE

		(* check for wildcard 'M' *)
		_nCharacterPosition := FIND(_sWildcard, 'M');
		IF _nCharacterPosition > 0 THEN

			(* generate month as 1 char and replace M *)
			_sData := arrMonthCode[stDateTime.wMonth];
			_sWildcard := REPLACE(_sWildcard, _sData, 1, _nCharacterPosition);
		END_IF
	END_IF

	(* insert strWildcard back into strInput *)
	F_STRING_Wildcard := INSERT(sString, _sWildcard, TO_INT(_fbExtractData.nStartPosition) - 1);

(* no wildcard string found *)
ELSE

	(* strInput direct to output without modification *)
	F_STRING_Wildcard := sString;
END_IF

END_FUNCTION

// Strings/Manipulation/F_STRING_WriteEscapeCharacters
(* Finds all instances of '&' in a given string and replaces it with it's escape character *)
FUNCTION F_STRING_WriteEscapeCharacters : T_MaxString
VAR_INPUT
	sString			: T_MaxString;		(* search string *)
END_VAR
VAR
	_nPosition		: UINT;
END_VAR

_nPosition := FIND(sString, '&');

IF _nPosition > 0 THEN

	F_STRING_WriteEscapeCharacters := REPLACE(sString, '&amp;',1 , _nPosition);

ELSE

	F_STRING_WriteEscapeCharacters := sString;

END_IF

END_FUNCTION

// Strings/Validation/F_STRING_InvalidateASCIIChar
(* checks a given string for characters that outside the range 0x21 -> 0x7A and 0x7C *)
FUNCTION F_STRING_InvalidateASCIIChar : INT
VAR_INPUT
	sString				: T_MaxString;		(* Search string *)
END_VAR
VAR
	_nCodeLen			: UINT;
	_nCharIndex			: UINT;
	_sCharacter			: T_Char;
END_VAR

(* reset output *)
F_STRING_InvalidateASCIIChar := 0;

(* strPackCode contains data *)
IF LEN(sString) = 0 THEN

	F_STRING_InvalidateASCIIChar := -1;

ELSIF LEN(sString) > 0 THEN

	(* check each char in the code *)
	FOR _nCharIndex := 1 TO LEN(sString) DO

		(* get char from string *)
		_sCharacter := MID(sString, 1, _nCharIndex);

		(* check if every character valid for proccessing *)
		IF (F_ToASC(_sCharacter) < 16#21 OR  F_ToASC(_sCharacter) >  16#7A) AND F_ToASC(_sCharacter) <> 16#7C THEN	(*  16#7C -> '|'*)

			(* update valid char counter *)
			F_STRING_InvalidateASCIIChar := F_STRING_InvalidateASCIIChar + 1;
			
		END_IF
		
	END_FOR
	
END_IF

END_FUNCTION

// Strings/Validation/F_STRING_InvalidateNumericChar
(* checks a given string for characters that outside the range 0x30 -> 0x39 *)
FUNCTION F_STRING_InvalidateNumericChar : INT
VAR_INPUT
	sString				: T_MaxString;
END_VAR
VAR
	_nCharacterIndex	: UINT;
	_sCharacter			: T_Char;
END_VAR

(* reset output *)
F_STRING_InvalidateNumericChar := 0;

(* strPackCode contains data *)
IF LEN(sString) > 0 THEN

	(* check each char in the code *)
	FOR _nCharacterIndex := 1 TO LEN(sString) DO

		(* get char from string *)
		_sCharacter := MID(sString, 1, _nCharacterIndex);

		(* check if every char valid for proccessig*)
		IF (F_ToASC(_sCharacter) < 16#30 OR  F_ToASC(_sCharacter) >  16#39) THEN

			(* update valid char counter *)
			F_STRING_InvalidateNumericChar := F_STRING_InvalidateNumericChar + 1;
			
		END_IF
		
	END_FOR
	
END_IF

END_FUNCTION

// Strings/Validation/F_STRING_IsNumber
(* returns true if the charachter is a number *)
FUNCTION F_STRING_IsNumber : BOOL
VAR_INPUT
	sCharacter			: T_Char; 		(* character to test *)
END_VAR
VAR
END_VAR

F_STRING_IsNumber := (F_ToASC(sCharacter) >= 16#30 AND F_ToASC(sCharacter) <= 16#39);

END_FUNCTION

// Strings/Validation/F_STRING_Validate
(* checks a string for various characteristics and returns a string if validation fails *)
FUNCTION F_STRING_Validate : T_MaxString
VAR_INPUT
	sString					: T_MaxString;	(* string to be examined *)
	nExpectedCharacters		: BYTE;			(* >0 = no of chars expected in string, 0 = chars not counted but string must not be empty *)
	nMaximumCharacters		: UINT;			(* >0 = max no of chars allowed in strFieldData, 0 = do not check *)
	bNumberCharactersOnly	: BOOL;			(* TRUE = all chars are checked to ensure only numerical (0-9) chars are present *)
	bDecimalPointAllowed	: BOOL;			(* TRUE = decimal point is allowed in a numerical string *)
END_VAR
VAR
	_nIndex					: UINT;
	_nCharacterValue		: BYTE;
END_VAR

(* string contains data *)
IF LEN(sString) > 0 THEN

	(* field data length exceeds specified maximum no of chars *)
	IF nMaximumCharacters > 0 AND LEN(sString) >= nMaximumCharacters THEN

		F_STRING_Validate := 'XML field data contains too many chars';

	(* string has expected no of chars OR string length does not matter *)
	ELSIF LEN(sString) = nExpectedCharacters OR nExpectedCharacters = 0 THEN

		(* string must only have numerical chars *)
		IF bNumberCharactersOnly THEN

			(* check each char in the string *)
			FOR _nIndex := 1 TO LEN(sString) DO

				(* convert char to ASCII value *)
				_nCharacterValue := F_ToASC(MID(sString, 1, _nIndex));

				(* string char is valid if 0-9, decimal point also allowed if enabled *)
				IF (_nCharacterValue >= F_ToASC('0') AND _nCharacterValue <= F_ToASC('9')) OR (_nCharacterValue = F_ToASC('.') AND bDecimalPointAllowed) THEN

					F_STRING_Validate := '';

				(* invalid char *)
				ELSE

					F_STRING_Validate := F_STRING_Concat3('Invalid char "', MID(sString, 1, _nIndex), '" found');
					EXIT;
					
				END_IF
				
			END_FOR

		(* string can be alpha-numeric chars *)
		ELSE

			F_STRING_Validate := '';
			
		END_IF

	(* string has incorrect no of chars *)
	ELSE

		F_STRING_Validate := F_STRING_Concat4('Expected length = ', BYTE_TO_STRING(nExpectedCharacters), ', actual length = ', INT_TO_STRING(LEN(sString)));

	END_IF

(* empty string *)
ELSE

	F_STRING_Validate := 'Empty';
	
END_IF

END_FUNCTION

// Strings/Validation/F_STRING_ValidateCode
(* checks a string for various characteristics and returns a code if validation fails *)
FUNCTION F_STRING_ValidateCode : E_STRING_ValidationCode
VAR_INPUT
	sString					: T_MaxString;	(* string to be examined *)
	nExpectedCharacters		: BYTE;			(* >0 = no of chars expected in string, 0 = chars not counted but string must not be empty *)
	nMaximumCharacters		: UINT;			(* >0 = max no of chars allowed in strFieldData, 0 = do not check *)
	bNumberCharactersOnly	: BOOL;			(* TRUE = all chars are checked to ensure only numerical (0-9) chars are present *)
	bDecimalPointAllowed	: BOOL;			(* TRUE = decimal point is allowed in a numerical string *)
END_VAR
VAR
	_nIndex					: UINT;
	_nCharacterValue		: BYTE;
END_VAR

(* string contains data *)
IF LEN(sString) > 0 THEN

	(* field data length exceeds specified maximum no of chars *)
	IF nMaximumCharacters > 0 AND LEN(sString) > nMaximumCharacters THEN

		F_STRING_ValidateCode := E_STRING_ValidationCode.MAXIMUM_LENGTH_EXCEEDED;

	(* string has expected no of chars OR string length does not matter *)
	ELSIF LEN(sString) = nExpectedCharacters OR nExpectedCharacters = 0 THEN

		(* string must only have numerical chars *)
		IF bNumberCharactersOnly THEN

			(* check each char in the string *)
			FOR _nIndex := 1 TO LEN(sString) DO

				(* convert char to ASCII value *)
				_nCharacterValue := F_ToASC(MID(sString, 1, _nIndex));

				(* string char is valid if 0-9, decimal point also allowed if enabled *)
				IF (_nCharacterValue >= F_ToASC('0') AND _nCharacterValue <= F_ToASC('9')) OR (_nCharacterValue = F_ToASC('.') AND bDecimalPointAllowed) THEN

					F_STRING_ValidateCode := E_STRING_ValidationCode.VALID;

				(* decimal point found but not allowed *)
				ELSIF _nCharacterValue = F_ToASC('.') AND bDecimalPointAllowed THEN

					F_STRING_ValidateCode := E_STRING_ValidationCode.INVALID_DECIMALPOINT;
					EXIT;

				(* other invalid char found *)
				ELSE

					F_STRING_ValidateCode := E_STRING_ValidationCode.INVALID;
					EXIT;
					
				END_IF
				
			END_FOR

		(* string can be alpha-numeric chars *)
		ELSE

			F_STRING_ValidateCode := E_STRING_ValidationCode.VALID;
			
		END_IF

	(* string is too short *)
	ELSIF LEN(sString) < nExpectedCharacters THEN

		F_STRING_ValidateCode := E_STRING_ValidationCode.TOO_SHORT;

	(* string is too long *)
	ELSIF LEN(sString) > nExpectedCharacters THEN

		F_STRING_ValidateCode := E_STRING_ValidationCode.TOO_LONG;
		
	END_IF

(* empty string *)
ELSE

	F_STRING_ValidateCode := E_STRING_ValidationCode.EMPTY_STRING;
	
END_IF

END_FUNCTION
